FUNCTION_BLOCK B_EQ_WSTRING (* Basic Function Block Type *)
  (* Standard: 61499-2 *)
  (* Version 0.0, 2016-02-15, 4DIAC-IDE, 4DIAC-Consortium *)
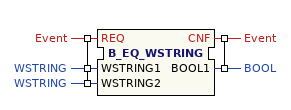
  EVENT_INPUT
    REQ WITH WSTRING1, WSTRING2; (* Normal Execution Request *)
  END_EVENT
  EVENT_OUTPUT
    CNF WITH BOOL1; (* Execution Confirmation *)
  END_EVENT
  VAR_INPUT
    WSTRING1 : WSTRING;
    WSTRING2 : WSTRING;
  END_VAR
  VAR_OUTPUT
    BOOL1 : BOOL := false;
  END_VAR
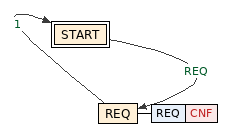
  EC_STATES
    START; (* Initial State *)
    REQ : REQ -> CNF; (* Normal execution *)
  END_STATES
  EC_TRANSITIONS
    START TO REQ := REQ;
    REQ TO START := 1;
  END_TRANSITIONS
  ALGORITHM REQ IN ST: (* Normally executed algorithm *)
IF WSTRING1= WSTRING2 THEN;
BOOL1:=TRUE;
ELSE
BOOL1:=FALSE;
END_IF;
  END_ALGORITHM
END_FUNCTION_BLOCK
